FUNCTION_BLOCK FB_TestMaschinentuer
VAR_INPUT
	bVentil : BOOL;
END_VAR
VAR_OUTPUT
	bDoorC : BOOL := TRUE;
	bDoorO : BOOL;
END_VAR
VAR
	RTrig : R_Trig;
	FTrig : F_Trig;
	fbTon1 : Ton;
	fbTon2 : Ton;
END_VAR

FTrig(CLK:= bVentil, Q=> );
RTrig(CLK:= bVentil, Q=> );
fbTon1(PT:= T#1S);
fbTon2(PT:= T#1S);

IF Ftrig.Q THEN
	fbTon1.IN := TRUE;
	bDoorC := FALSE;
END_IF
	IF fbTon1.Q THEN
		bDoorO := TRUE;
		fbTon1.IN := FALSE;
	END_IF



IF RTrig.Q THEN
	fbTon2.In := TRUE;
	bDoorO := FALSE;
END_IF
	IF fbTon2.Q THEN
		bDoorC := TRUE;
		fbTon2.IN := FALSE;
	END_IF

END_FUNCTION_BLOCK

(* stored: Version 1.1.0.1, ProductVersion 3.1.4024.15
   POU FB_TestMaschinentuer: Id {ab01a79a-aada-4046-9f2b-8940044b684c}, SpecialFunc None *)
